TYPE E_TankState :
(	TANK_IDLE := 0,
	TANK_STOP := 5,
	TANK_WITHDRAWING := 10,
	TANK_FILLING:= 20
);
END_TYPE

(* stored: Version 1.1.0.1, ProductVersion 3.1.4024.12
   DUT E_TankState: Id {625f87ac-beaf-43c0-b351-9d294cfb9376} *)
